(* IEC 61131-3 sources: CodesysTest/alpha/export/Pro18_1174_04.dev/Plc Logic/Application/Motors/Applied Motion/DataHandlers, 2 files *)

(* ---- FB_StepServoAlarms.pou.st ---- *)
(*#-#-#-#-#-#-#-#-#-#---Declaration---#-#-#-#-#-#-#-#-#-#-#-#-#*)

FUNCTION_BLOCK FB_StepServoAlarms
VAR_INPUT
    alarmCode : INT;
END_VAR
VAR_OUTPUT
    positionLimit : BOOL;        // FAULT - Motor exceeded position limit - following error
    CCWLimit : BOOL;      // WARNING - Motor is at CCW Limit
    CWLimit : BOOL;      // WARNING - Motor is at CW Limit
    overTemp : BOOL;      // FAULT - Motor Over Temperature Limit
    internalVoltage : BOOL;      // FAULT - Internal Voltage Fault
    overVoltage    : BOOL;      // FAULT - Overvoltage Fault
    underVoltage : BOOL;      // WARNING - Undervoltage Warning
    overCurrent : BOOL;      // FAULT - Motor Overcurrent
    openMotorWinding : BOOL;      // FAULT - Motor Detected Open Winding
    badEncoder : BOOL;      // FAULT - Motor Encoder Failure
    commError : BOOL;      // WARNING - Communications Error
    badFlash : BOOL;      // WARNING - Bad Flash
    noMove : BOOL;      // WARNING - No Move
    currentFoldback    : BOOL;      // WARNING - Current Foldback
    blankQSegment : BOOL;      // WARNING - Blank Q Segment
    NVMemoryDoubleError : BOOL;      // WARNING - NV Memory Double Error
END_VAR
VAR
END_VAR
VAR_IN_OUT
	faults : StepServoFaultsType;
END_VAR(*#-#-#-#-#-#-#-#-#-#---Implementation---#-#-#-#-#-#-#-#-#-#-#-#-#*)

//    Fucntion Block: FB_StepServoAlarms
//    Description: This unpacks the step servo alarm bits from the alarm word received over EIP
//    Created by: Ben Hess
//    Created Date: September 5th, 2018

faults.positionLimit.faultTrigger := positionLimit := alarmCode.0;
faults.CCWLimit.faultTrigger := CCWLimit := alarmCode.1;
faults.CWLimit.faultTrigger := CWLimit := alarmCode.2;
faults.overTemp.faultTrigger := overTemp := alarmCode.3;
faults.internalVoltage.faultTrigger := internalVoltage := alarmCode.4;
faults.overVoltage.faultTrigger := overVoltage := alarmCode.5;
faults.underVoltage.faultTrigger := underVoltage := alarmCode.6;
faults.overCurrent.faultTrigger := overCurrent := alarmCode.7;
faults.openMotorWinding.faultTrigger := openMotorWinding := alarmCode.8;
faults.badEncoder.faultTrigger := badEncoder := alarmCode.9;
commError := alarmCode.10;
badFlash := alarmCode.11;
faults.noMove.faultTrigger := noMove := alarmCode.12;
faults.currentFoldback.faultTrigger := currentFoldback := alarmCode.13;
blankQSegment := alarmCode.14;
NVMemoryDoubleError := alarmCode.15;

(* ---- StepServoStatusFB.pou.st ---- *)
(*#-#-#-#-#-#-#-#-#-#---Declaration---#-#-#-#-#-#-#-#-#-#-#-#-#*)

FUNCTION_BLOCK StepServoStatusFB
VAR_INPUT
    statusCode : INT;
END_VAR
VAR_OUTPUT
    motorEnabled : BOOL;        //Motor Enabled (Motor Disabled if this bit = 0)
    sampling : BOOL;      //Sampling (for Quick Tuner)
    driveFaulted : BOOL;      //Drive Fault (check Alarm Code)
    inPosition : BOOL;      //In Position (motor is in position)
    moving : BOOL;      //Moving (motor is moving)
    jogging    : BOOL;      //Jogging (currently in jog mode)
    stopping : BOOL;      //Stopping (in the process of stopping from a stop command)
    waitingForInput : BOOL;      //Waiting (for an input; executing a WI command)
    saving : BOOL;      //Saving (parameter data is being saved)
    alarmPresent : BOOL;      //Alarm present (check Alarm Code)
    homing : BOOL;      //Homing (executing an SH command)
    waitingForTime : BOOL;      //Waiting (for time; executing a WD or WT command)
    wizardRunning : BOOL;      //Wizard running (Timing Wizard is running)
    checkingEncoder    : BOOL;      //Checking encoder (Timing Wizard is running)
    Q_ProgramRunning : BOOL;      //Q Program is running
    initializing : BOOL;      //Initializing (happens at power up) ; Servo Ready (for SV200 drives only)
END_VAR
VAR
END_VAR
(*#-#-#-#-#-#-#-#-#-#---Implementation---#-#-#-#-#-#-#-#-#-#-#-#-#*)

//    Fucntion Block: StepServoStatus
//    Description: This unpacks the step servo status bits from the status word received over modbus
//    Created by: Ben Hess
//    Created Date: January 26th, 2018

motorEnabled := statusCode.0;
sampling := statusCode.1;
driveFaulted := statusCode.2;
inPosition := statusCode.3;
moving := statusCode.4;
jogging := statusCode.5;
stopping := statusCode.6;
waitingForInput    := statusCode.7;
saving := statusCode.8;
alarmPresent := statusCode.9;
homing := statusCode.10;
waitingForTime := statusCode.11;
wizardRunning := statusCode.12;
checkingEncoder := statusCode.13;
Q_ProgramRunning := statusCode.14;
initializing := statusCode.15;
